FUNCTION_BLOCK AX2_BOOL_TO_X (* Composite FB for convert BOOL to AX2 *)
  (* Standard: 61499-2; Description: Copyright (c) 2024 HR Agrartechnik GmbH This program and the accompanying materials are made available under the terms of the Eclipse Public License 2.0 which is available at https://www.eclipse.org/legal/epl-2.0/ SPDX-License-Identifier: EPL-2.0 *)
  (* Version 1.0, 2024-04-24, Franz Höpfinger, HR Agrartechnik GmbH *)
  PACKAGE adapter::conversion::bidirectional;
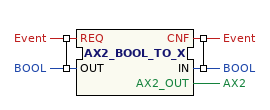
  EVENT_INPUT
    REQ WITH OUT; (* Request to Adapter *)
  END_EVENT
  EVENT_OUTPUT
    CNF WITH IN; (* Confirmation from Adapter *)
  END_EVENT
  VAR_INPUT
    OUT : BOOL;
  END_VAR
  VAR_OUTPUT
    IN : BOOL; (* Input data from Adapter *)
  END_VAR
  PLUGS
    AX2_OUT : adapter::types::bidirectional::AX2; (* Adapter Output *)
  END_PLUGS
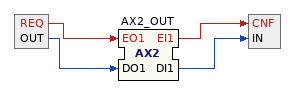
  EVENT_CONNECTIONS
    REQ TO AX2_OUT.EO1;
    AX2_OUT.EI1 TO CNF;
  END_CONNECTIONS
  DATA_CONNECTIONS
    OUT TO AX2_OUT.DO1;
    AX2_OUT.DI1 TO IN;
  END_CONNECTIONS
END_FUNCTION_BLOCK
